FUNCTION_BLOCK FB_DI (* Service Interface Function Block Type *)
  (* Standard: 61499-2 *)
  (* Version 0.0, 2014-5-4, wildai, nxtControl GmbH, template *)
  (* Compiler Cpp nxtControl builtin 1.0 *)
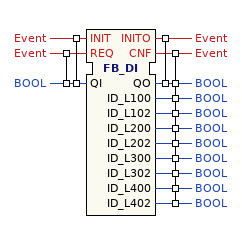
  EVENT_INPUT
    INIT WITH QI; (* Service Initialization *)
    REQ WITH QI; (* Service Request *)
  END_EVENT
  EVENT_OUTPUT
    INITO WITH QO; (* Initialization Confirm *)
    CNF WITH QO, ID_L100, ID_L102, ID_L200, ID_L202, ID_L300, ID_L302, ID_L400, ID_L402; (* Confirmation of Requested Service *)
  END_EVENT
  VAR_INPUT
    QI : BOOL; (* Event Input Qualifier *)
  END_VAR
  VAR_OUTPUT
    QO : BOOL; (* Event Output Qualifier *)
    ID_L100 : BOOL; (* Input data from resource *)
    ID_L102 : BOOL;
    ID_L200 : BOOL;
    ID_L202 : BOOL;
    ID_L300 : BOOL;
    ID_L302 : BOOL;
    ID_L400 : BOOL;
    ID_L402 : BOOL;
  END_VAR
  SERVICE FB_DI/RESOURCE
    SEQUENCE normal_establishment
      FB_DI.INIT+(PARAMS) -> RESOURCE.initialize(PARAMS) -> FB_DI.INITO+();
    END_SEQUENCE
    SEQUENCE unsuccessful_establishment
      FB_DI.INIT+(PARAMS) -> RESOURCE.initialize(PARAMS) -> FB_DI.INITO-(STATUS);
    END_SEQUENCE
    SEQUENCE request_confirm
      FB_DI.REQ+(SD) -> RESOURCE.request(SD) -> FB_DI.CNF+(RD);
    END_SEQUENCE
    SEQUENCE request_inhibited
      FB_DI.REQ-(SD) -> FB_DI.CNF-(STATUS);
    END_SEQUENCE
    SEQUENCE request_error
      FB_DI.REQ+(SD) -> RESOURCE.request(SD) -> FB_DI.CNF-(STATUS);
    END_SEQUENCE
    SEQUENCE indication_response
      FB_DI.RSP(QI,SD) -> RESOURCE.response(QI,SD);
      RESOURCE.indicate(RD) -> FB_DI.IND+(RD);
    END_SEQUENCE
    SEQUENCE indication_inhibited
      RESOURCE.indicate(RD,QI=FALSE) -> RESOURCE.inhibited();
    END_SEQUENCE
    SEQUENCE error_indication
      RESOURCE.error(STATUS) -> FB_DI.IND-(STATUS);
    END_SEQUENCE
    SEQUENCE application_initiated_termination
      FB_DI.INIT-() -> RESOURCE.terminate() -> FB_DI.INITO-(STATUS);
    END_SEQUENCE
    SEQUENCE resource_initiated_termination
      -> FB_DI.INITO-(STATUS);
    END_SEQUENCE
  END_SERVICE
END_FUNCTION_BLOCK
